(* PLC project Unnamed, Unknown Unnamed 1 *)
(* stored: creationDateTime 2026-06-15T08:02:50, modificationDateTime 2026-06-15T08:02:50 *)

FUNCTION SUMN : ANY_NUM
  VAR_INPUT
    IN1 : ANY_NUM;
    IN2 : ANY_NUM;
  END_VAR

END_FUNCTION

PROGRAM PLC_PRG
  VAR
    a : INT;
    b : INT;
    c : INT;
    result : INT;
  END_VAR

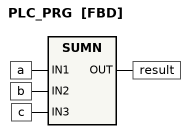
(* FBD diagram, written out as Structured Text *)
result := SUMN(a, b, c);
END_PROGRAM

CONFIGURATION Config0
  RESOURCE Res0 ON PLC
    TASK task0(INTERVAL := T#20ms, PRIORITY := 1);
    PROGRAM instance0 WITH task0 : PLC_PRG;
  END_RESOURCE
END_CONFIGURATION
